INTERFACE I_Extensions

METHOD PUBLIC Accept
VAR_INPUT
	Visitor : I_ExtensionVisitor;
END_VAR
END_METHOD

METHOD AddExtension
VAR_INPUT
	Extension : I_Extension;
END_VAR
END_METHOD

METHOD PUBLIC TryGetExtensionByName : BOOL
VAR_INPUT
	Name : T_MAXSTRING;
	Destination : REFERENCE TO I_Extension;
END_VAR
END_METHOD

END_INTERFACE

(* stored: Version 1.1.0.1, ProductVersion 3.1.4024.12
   Itf I_Extensions: Id {7db66379-e861-4d2c-a5d6-50c9090adb8f}
   Method Accept: Id {ed7ca7fe-c97f-4965-aab1-6b8e2c9438db}
   Method AddExtension: Id {3e68d2ee-2c9a-4e4f-8ad4-40deaaf44331}
   Method TryGetExtensionByName: Id {5b8e704e-81bf-4c64-a676-068e39f90b17} *)
